% RSLogix 500 project CHEMICAL MIXING PROCESS_BAK004.RSS, saved by version 8.30.00.16 %
PROJECT "UNTITLED"    % processor: Bul.1763 MicroLogix 1100 Series B %

PROGRAM FILES
  LAD 2   8 rungs

DATA FILES
  O0 OUTPUT  4 elements
  I1 INPUT  6 elements
  S2 STATUS  66 elements
  B3 BINARY  1 elements
  T4 TIMER  1 elements
  C5 COUNTER  1 elements
  R6 CONTROL  1 elements
  N7 INTEGER  1 elements
  F8 FLOAT  1 elements

LADDER 2
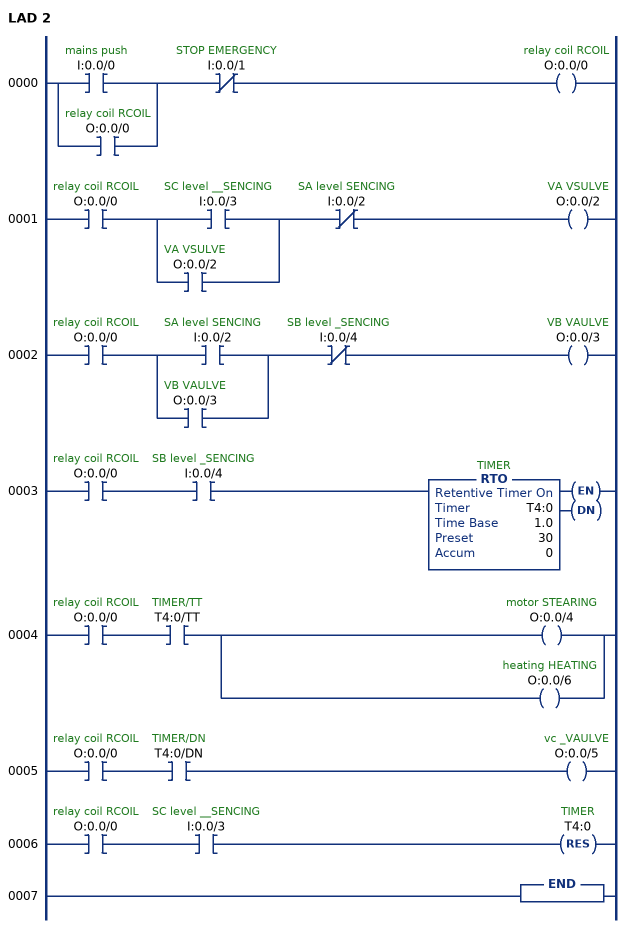
% Rung: 0 %
SOR BST XIC I:0.0/0 NXB XIC O:0.0/0 BND XIO I:0.0/1 OTE O:0.0/0 EOR
%   I:0.0/0  "mains push" %
%   O:0.0/0  RCOIL  "relay coil" %
%   I:0.0/1  EMERGENCY  "STOP" %
% Rung: 1 %
SOR XIC O:0.0/0 BST XIC I:0.0/3 NXB XIC O:0.0/2 BND XIO I:0.0/2 OTE O:0.0/2 EOR
%   O:0.0/0  RCOIL  "relay coil" %
%   I:0.0/3  __SENCING  "SC level" %
%   O:0.0/2  VSULVE  "VA" %
%   I:0.0/2  SENCING  "SA level" %
% Rung: 2 %
SOR XIC O:0.0/0 BST XIC I:0.0/2 NXB XIC O:0.0/3 BND XIO I:0.0/4 OTE O:0.0/3 EOR
%   O:0.0/0  RCOIL  "relay coil" %
%   I:0.0/2  SENCING  "SA level" %
%   O:0.0/3  VAULVE  "VB" %
%   I:0.0/4  _SENCING  "SB level" %
% Rung: 3 %
SOR XIC O:0.0/0 XIC I:0.0/4 RTO T4:0 1.0 30 0 EOR
%   O:0.0/0  RCOIL  "relay coil" %
%   I:0.0/4  _SENCING  "SB level" %
%   T4:0  TIMER %
% Rung: 4 %
SOR XIC O:0.0/0 XIC T4:0/TT BST OTE O:0.0/4 NXB OTE O:0.0/6 BND EOR
%   O:0.0/0  RCOIL  "relay coil" %
%   T4:0  TIMER %
%   O:0.0/4  STEARING  "motor" %
%   O:0.0/6  HEATING  "heating" %
% Rung: 5 %
SOR XIC O:0.0/0 XIC T4:0/DN OTE O:0.0/5 EOR
%   O:0.0/0  RCOIL  "relay coil" %
%   T4:0  TIMER %
%   O:0.0/5  _VAULVE  "vc" %
% Rung: 6 %
SOR XIC O:0.0/0 XIC I:0.0/3 RES T4:0 EOR
%   O:0.0/0  RCOIL  "relay coil" %
%   I:0.0/3  __SENCING  "SC level" %
%   T4:0  TIMER %
% Rung: 7 %
SOR END EOR

DATA TABLE (non-zero values as saved)
DATA T4
% .PRE .ACC %
% T4:0 % 30 0
